PROGRAM CommWithPC
VAR
END_VAR

END_PROGRAM

(* stored: Version 1.1.0.1, ProductVersion 3.1.4024.9
   POU CommWithPC: Id {bac48c79-57e4-4fc5-9e09-7581a510d3e9}, SpecialFunc None *)
